(*
    TcXunit interpreter fixture (TcXunit-p3t.4). Suite whose test method
    faults inside FB_FailingLineHelper: the reported location must be the
    INNERMOST body's POU/method/line, not this suite's call site.
*)
FUNCTION_BLOCK FB_FailingLineTests EXTENDS TcUnit.FB_TestSuite
VAR
	helper : FB_FailingLineHelper;
END_VAR

FaultsDeepInAHelper();

METHOD PRIVATE FaultsDeepInAHelper
TEST('FaultsDeepInAHelper');

(* Caller-side call site: NOT the line the failure log should name. *)
helper.ThrowsFromNestedCall();

TEST_FINISHED();
END_METHOD

END_FUNCTION_BLOCK

(* stored: Version 1.1.0.1, ProductVersion 3.1.4026.18
   POU FB_FailingLineTests: Id {c4d5e6f7-0004-4a1a-8b1b-000000000003}, SpecialFunc None
   Method FaultsDeepInAHelper: Id {c4d5e6f7-0004-4a1a-8b1b-000000000004} *)
